// TIA Portal V20 export
TYPE "LWONIK_typeZoneStatus"
// stored: Access Published
   STRUCT
      safetyReleased1 : Bool;
      safetyReleased2 : Bool;
      ackReq : Bool;
      safetyFault : Bool;
      highSpeedEnable : Bool;
      activeSLS : Bool;
      activeSTO : Bool;
      activeSOS : Bool;
      activeSS1 : Bool;
      activeSS2 : Bool;
      AllFDoorClose : Bool;
      SFDoorOpen : Bool;
      MFDoorOpen : Bool;
   END_STRUCT;
END_TYPE
